PROGRAM PRG_TEST
VAR
	foo:FB_EventBuffer_Test;	



END_VAR

TcUnit.RUN();

END_PROGRAM

(* stored: Version 1.1.0.1, ProductVersion 3.1.4024.12
   POU PRG_TEST: Id {11123ccf-6161-4104-a105-7a5ea8ba132b}, SpecialFunc None *)
